Staubli VAL3: DECTOBIN.pgx

public program decToBin(num x_value, string& x_return[])
// change num variable to binary string (e.g. 9 => "1001")
  local num l_bit
  local num l_value
  local num l_mask
begin
  l_mask=0
  l_bit=1
  x_return=""
  l_value=roundDown(x_value)
  do
    call bmask(l_bit,l_mask)
    if (l_value%2)==0
      x_return="0"+x_return
    else
      x_return="1"+x_return
    endIf
    l_value=roundDown(l_value/2)
    l_bit=l_bit+1
  until l_mask>x_value
  if bDebug
    putln("decToBin(): "+toString("0.0",x_value)+" => "+x_return)
  endIf
end
